FUNCTION_BLOCK Test_ReadBySymbolName EXTENDS TUnitTestBase
VAR
    AdsReadBySymbolName : TAdsReadBySymbolName;
    ValueToRead : INT;
    ReadResult  : INT;
    ScanCount : DINT;
    State: INT;
END_VAR

CASE State OF
    0:
        ValueToRead := 1234;
        ReadResult := 0;
        ScanCount := 0;
    
        AdsReadBySymbolName.Execute(
            AmsNetId:= '', 
            Port:= 851, 
            SymbolName:= 'PB_TestRunner.Test_ReadBySymbolName.ValueToRead', 
            ReadDataAddress:= ADR(ReadResult), 
            ReadDataLength:= SIZEOF(ReadResult), 
            KeepSymbolHandle:= FALSE);

        State := 10;
        
    10:
        ScanCount := ScanCount + 1;
        IF NOT AdsReadBySymbolName.Execution.Busy THEN
            State := 20;    
		END_IF
        
    20:
        Assertion.AssertEquals_INT(
            Expected     := 1234,
            Actual       := ReadResult,
            ObjectName   := _TestName,
            Variablename := 'ReadResult'); 
 
        TestFinished();
        State := 0;
END_CASE

AdsReadBySymbolName();

END_FUNCTION_BLOCK

(* stored: Version 1.1.0.1, ProductVersion 3.1.4024.3
   POU Test_ReadBySymbolName: Id {78aa2181-6b0e-0a51-1703-22792cf8286e}, SpecialFunc None *)
